PROGRAM P_ControlBlock
VAR
	fbControlBlock : FB_ControlBlock;
END_VAR

fbControlBlock(
	ssMethodType := BOOL_TO_SINT(G_VirtualControlBox.bGreenLight),
	X_real:= G_Sensors.fPistonPosition,
	Pa:= G_Sensors.fPressurePistonSide, 
	Pb := G_Sensors.fPressureRodSide,
	Ps:= G_Sensors.fPressureSupply,
	Clock := 1,
	u	=> G_Work.fControlOutputNormalized
);

END_PROGRAM

(* stored: Version 1.1.0.1, ProductVersion 3.1.4024.13
   POU P_ControlBlock: Id {1c742f8d-99bf-4aa1-ba99-fa370ccce2ab}, SpecialFunc None *)
